TYPE ST_HW_InputsTurnTable :

STRUCT
	TT						: ST_HW_InputsTT; //Turning inputs	
	//Drive/Transport control sensors
	Sensor_Stop_12			: BOOL; // Sensor stop axis 1-2 forward
	Sensor_Creep_12			: BOOL; // Sensor creep speed axis 1-2 forward	
	Sensor_Stop_21			: BOOL; // Sensor stop axis 1-2 reverse	
	Sensor_Creep_21			: BOOL; // Sensor creep speed axis 1-2 reverse
	
	Sensor_Overhang_12		: BOOL; // Sensor overhang axis 1-2 forward	
	Sensor_Overhang_21		: BOOL; // Sensor overhang axis 2-1 reverse				
END_STRUCT
END_TYPE

(* stored: Version 1.1.0.1, ProductVersion 3.1.4024.9
   DUT ST_HW_InputsTurnTable: Id {3e7e84ad-a0c9-4042-9587-636df92fcea6} *)
